{attribute 'c++_compatible'}
///Standard cylinder
INTERFACE I_StandardCylinder EXTENDS I_Object

///Cylinder at home position
PROPERTY AtHome : BOOL
GET
END_GET
END_PROPERTY

///Cylinder at out position
PROPERTY AtOut : BOOL
GET
END_GET
END_PROPERTY

///Enable cylinder to change position
PROPERTY Enable : BOOL
GET
END_GET
SET
END_SET
END_PROPERTY

METHOD MoveHome
VAR_INPUT
END_VAR
END_METHOD

METHOD MoveOut
VAR_INPUT
END_VAR
END_METHOD

///Pointer to settings, should be set at FB_init but can be modified with set accessor if needed
PROPERTY Settings : POINTER TO ST_StandardCylinderSettings
GET
END_GET
SET
END_SET
END_PROPERTY

END_INTERFACE

(* stored: Version 1.1.0.1, ProductVersion 3.1.4019.2
   Itf I_StandardCylinder: Id {d18b866f-0390-430e-9b9e-caee21315be4}
   Folder Settings: Id {8b07865b-2db7-4e1e-aace-a3fe3af82c1c}
   Property AtHome: Id {25d96ad8-4fa5-4096-879f-88b8c60bddcc}
   Get Get: Id {511eb874-2f63-4231-b605-17869733e443}
   Property AtOut: Id {fadbb3b1-5440-45fe-a196-e2780bda1083}
   Get Get: Id {16dafb83-1e25-4c40-899e-33887945afd6}
   Property Enable: Id {45e19fc6-373e-42b3-8802-a5d94e051cce}
   Get Get: Id {e06bb2c9-1bca-46c2-ad0f-f41259df3160}
   Set Set: Id {c1e0ad01-c59c-4e35-b89d-121c06ea65fc}
   Method MoveHome: Id {104230db-bc98-464b-85e4-52736146d9ab}
   Method MoveOut: Id {f79ad045-0a6d-4a0f-9730-f5b646040f70}
   Property Settings: Id {2bd5fba4-139c-45c4-949d-2bddd597fc2b}
   Get Get: Id {00185921-0d47-46f2-985a-6b44282f4bd0}
   Set Set: Id {f9d2d5be-559c-4028-83ee-802b1f1565c8} *)
